PROGRAM PRG_TEST
VAR
	//fb_SL3K4ReadPMPSDB_Test : FB_SL3K4ReadPMPSDB_Test;
	//fb_SL3K4_Test : FB_SL3K4_Test;
	//fb_SL3K4BPTM_Test : FB_SL3K4BPTM_Test;
	//fb_DGPD_Test : FB_DGPD_Test;
	//fb_SequenceMover_Test : FB_SequenceMover_Test;
	//fb_DGPDEPS_Test :  FB_DGPDEPS_Test;
END_VAR

TcUnit.Run();

END_PROGRAM

(* stored: Version 1.1.0.1
   POU PRG_TEST: Id {a023bf89-c141-4a93-8485-ae7e96fe0db6}, SpecialFunc None *)
